Staubli VAL3: setTool.pgx

public program setTool(tool tParGun, num x_nIndex)
begin
  saveTool:gun[x_nIndex].trsf=tParGun.trsf
end
